{attribute addProperty BoxType "EL3692-0000-0017"}
{attribute addProperty Id "UnderrangeBIT10.1251OverrangeBIT10.1252Extended_rangeBIT10.1253Data_invalidBIT10.1254Range_invalidBIT10.1255Autorange_disabledBIT10.1256ErrorBIT10.1257Steady_stateBIT10.1259TxPDO_StateBIT10.1257TxPDO_ToggleBIT10.1259"}
{attribute addProperty CRC "2290965246"}
{attribute addProperty SizeInBites "16"}
{attribute addProperty SizeInBytes "2"}
TYPE Status_888D5AFE :
STRUCT
	{attribute addProperty Name "Underrange"}
	Underrange : BIT;
	{attribute addProperty Name "Overrange"}
	Overrange : BIT;
	{attribute addProperty Name "Extended_range"}
	Extended_range : BIT;
	{attribute addProperty Name "Data_invalid"}
	Data_invalid : BIT;
	{attribute addProperty Name "Range_invalid"}
	Range_invalid : BIT;
	{attribute addProperty Name "Autorange_disabled"}
	Autorange_disabled : BIT;
	{attribute addProperty Name "Error"}
	Error : BIT;
	{attribute 'hide'}
	reserve_1 : BIT;
	{attribute addProperty Name "Steady_state"}
	Steady_state : BIT;
	{attribute 'hide'}
	reserve_2_BIT_0 : BIT;
	{attribute 'hide'}
	reserve_2_BIT_1 : BIT;
	{attribute 'hide'}
	reserve_2_BIT_2 : BIT;
	{attribute 'hide'}
	reserve_2_BIT_3 : BIT;
	{attribute 'hide'}
	reserve_2_BIT_4 : BIT;
	{attribute addProperty Name "TxPDO_State"}
	TxPDO_State : BIT;
	{attribute addProperty Name "TxPDO_Toggle"}
	TxPDO_Toggle : BIT;
END_STRUCT
END_TYPE

(* stored: Version 1.2.0.0, ProductVersion 3.1.4024.9
   DUT Status_888D5AFE: Id {53bca0ad-9547-4ac1-b87d-37c072a5e822} *)
